INTERFACE ITF_EM_Seal_Shrink

END_INTERFACE

(* stored: Version 1.1.0.1, ProductVersion 3.1.4024.12
   Itf ITF_EM_Seal_Shrink: Id {426d6fb7-c3a7-49e5-96ef-dad5f5903895} *)
